{attribute addProperty BoxType "EL2819-0000-0016"}
{attribute addProperty Id "ChannelAT %Q*ARRAY[0 ..15] OF Channel_D3FEAEF91620"}
{attribute addProperty CRC "3516801023"}
{attribute addProperty SizeInBites "16"}
{attribute addProperty SizeInBytes "2"}
TYPE DIG_Outputs_FCF3AB2C :
STRUCT
	{attribute addProperty Name "Channel"}
	Channel AT %Q* : ARRAY[0 ..15] OF Channel_D3FEAEF9;
END_STRUCT
END_TYPE

(* stored: Version 1.2.0.0, ProductVersion 3.1.4024.9
   DUT DIG_Outputs_FCF3AB2C: Id {86e878b7-9e1c-4974-8029-b620fbd8537e} *)
